// TIA Portal V20 export
TYPE "UDT_Service_DintServParam"
   STRUCT
      OSLevel : Byte;
      ApplyExt : Bool;
      ApplyOp : Bool;
      Sync : Bool;
      StateOffOp : Bool;
      StateOpOp : Bool;
      StateAutOp : Bool;
      SrcIntOp : Bool;
      SrcExtOp : Bool;
      VExt : DInt;
      VOp : DInt;
   END_STRUCT;
END_TYPE
